SYSTEM FillerModule (* Module Filler, generated from its module specification *)
  (* Standard: 61499-2 *)
  APPLICATION Filler (* Module Filler on target pc (localhost, IO modbus; generated by modgen) *)
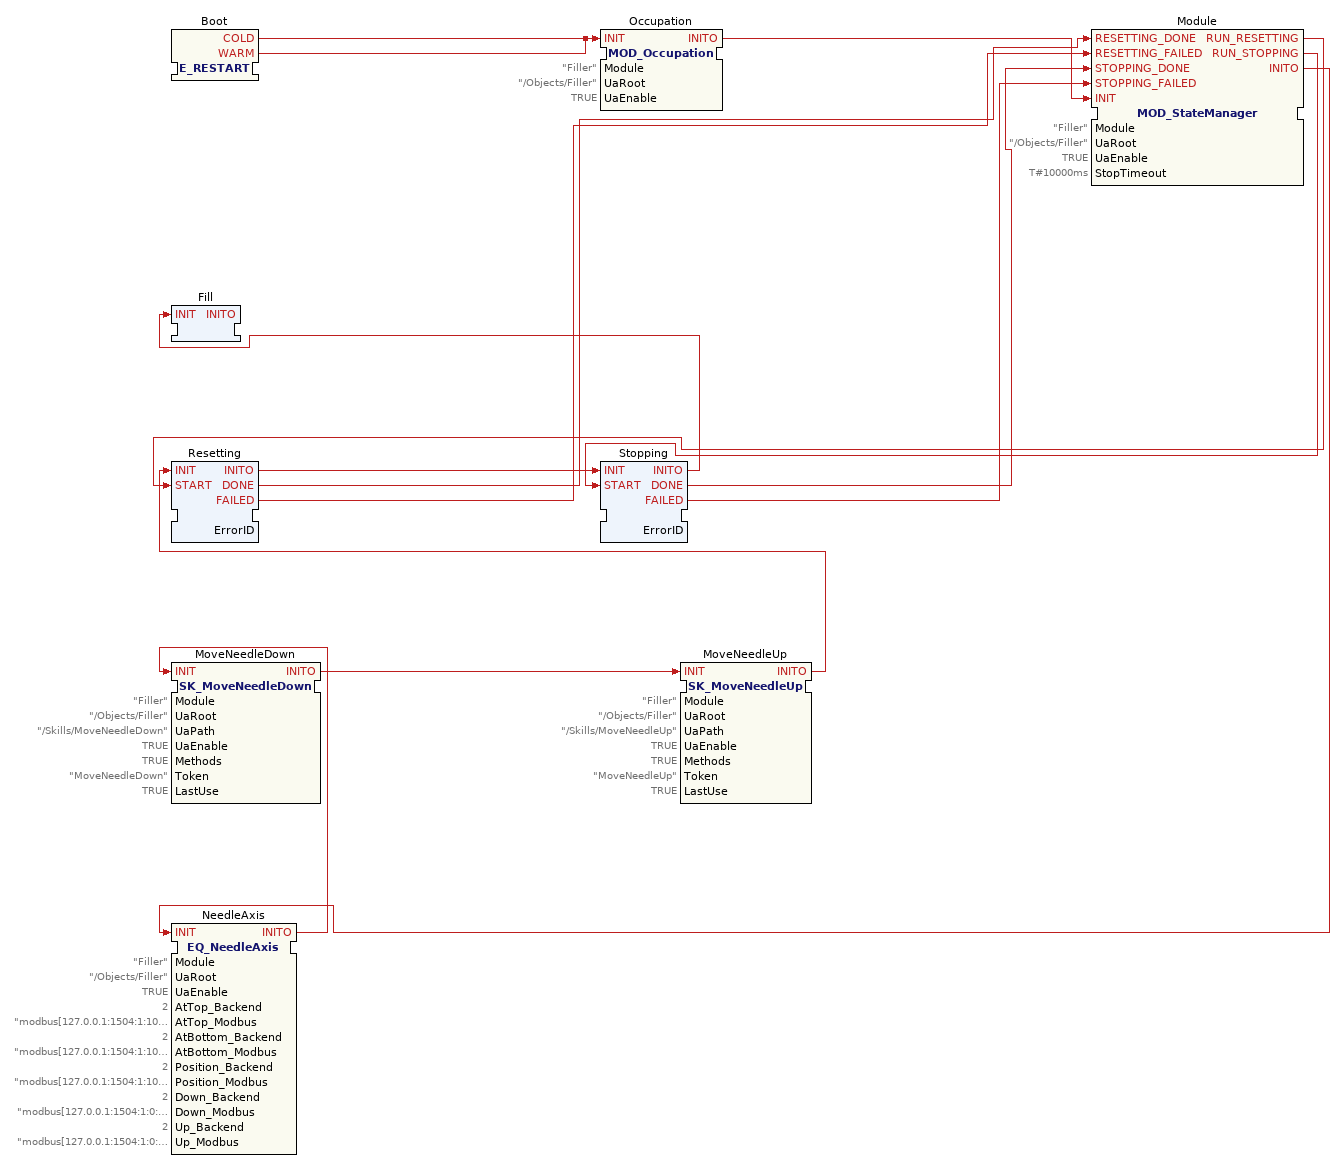
    (* Group ModuleLevel: Module level: occupation, PackML state manager, start-up and the target's IO lines *)
    (* Group ModuleLevelSkills: Module level skills: Control, Sequences (Execute, Stop) of skill primitives and Release; OPC UA /Skills/<name> *)
    (* Group Procedures: Procedures the module state manager runs while Resetting and Stopping *)
    (* Group SkillPrimitives: Skill primitives: one equipment command until a sensor or a time; OPC UA /Skills/<name> *)
    (* Group EquipmentIO: Equipment IO: the only owners of the IO points; skills send them output values over local channels *)
    FBS
      Boot : iec61499::events::E_RESTART; {SET_ATTRIBUTE(GroupName, ModuleLevel)}
      Occupation : modlib::MOD_Occupation(Module := "Filler", UaRoot := "/Objects/Filler", UaEnable := TRUE); {SET_ATTRIBUTE(GroupName, ModuleLevel)}
      Module : modlib::MOD_StateManager(Module := "Filler", UaRoot := "/Objects/Filler", UaEnable := TRUE, StopTimeout := T#10000ms); {SET_ATTRIBUTE(GroupName, ModuleLevel)}
      NeedleAxis : filler::EQ_NeedleAxis(Module := "Filler", UaRoot := "/Objects/Filler", UaEnable := TRUE, AtTop_Backend := 2, AtTop_Modbus := "modbus[127.0.0.1:1504:1:10:d0:]", AtBottom_Backend := 2, AtBottom_Modbus := "modbus[127.0.0.1:1504:1:10:d1:]", Position_Backend := 2, Position_Modbus := "modbus[127.0.0.1:1504:1:10:i1:]", Down_Backend := 2, Down_Modbus := "modbus[127.0.0.1:1504:1:0::c0]", Up_Backend := 2, Up_Modbus := "modbus[127.0.0.1:1504:1:0::c2]"); {SET_ATTRIBUTE(GroupName, EquipmentIO)}
      MoveNeedleDown : filler::SK_MoveNeedleDown(Module := "Filler", UaRoot := "/Objects/Filler", UaPath := "/Skills/MoveNeedleDown", UaEnable := TRUE, Methods := TRUE, Token := "MoveNeedleDown", LastUse := TRUE); {SET_ATTRIBUTE(GroupName, SkillPrimitives)}
      MoveNeedleUp : filler::SK_MoveNeedleUp(Module := "Filler", UaRoot := "/Objects/Filler", UaPath := "/Skills/MoveNeedleUp", UaEnable := TRUE, Methods := TRUE, Token := "MoveNeedleUp", LastUse := TRUE); {SET_ATTRIBUTE(GroupName, SkillPrimitives)}
    END_FBS
    SUBAPPLICATION Resetting (* Procedure the module runs while Resetting *)
      {SET_ATTRIBUTE(GroupName, Procedures)}
      EVENT_INPUT
        INIT : EInit;
        START;
      END_EVENT
      EVENT_OUTPUT
        INITO : EInit;
        DONE;
        FAILED;
      END_EVENT
      VAR_OUTPUT
        ErrorID : UINT;
      END_VAR
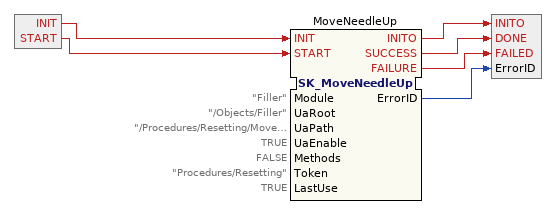
      FBS
        MoveNeedleUp : filler::SK_MoveNeedleUp(Module := "Filler", UaRoot := "/Objects/Filler", UaPath := "/Procedures/Resetting/MoveNeedleUp", UaEnable := TRUE, Methods := FALSE, Token := "Procedures/Resetting", LastUse := TRUE);
      END_FBS
      EVENT_CONNECTIONS
        INIT TO MoveNeedleUp.INIT;
        MoveNeedleUp.INITO TO INITO;
        START TO MoveNeedleUp.START;
        MoveNeedleUp.SUCCESS TO DONE;
        MoveNeedleUp.FAILURE TO FAILED;
      END_CONNECTIONS
      DATA_CONNECTIONS
        MoveNeedleUp.ErrorID TO ErrorID;
      END_CONNECTIONS
    END_SUBAPPLICATION
    SUBAPPLICATION Stopping (* Procedure the module runs while Stopping *)
      {SET_ATTRIBUTE(GroupName, Procedures)}
      EVENT_INPUT
        INIT : EInit;
        START;
      END_EVENT
      EVENT_OUTPUT
        INITO : EInit;
        DONE;
        FAILED;
      END_EVENT
      VAR_OUTPUT
        ErrorID : UINT;
      END_VAR
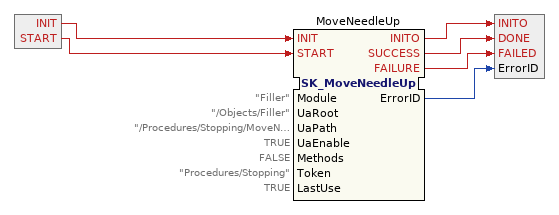
      FBS
        MoveNeedleUp : filler::SK_MoveNeedleUp(Module := "Filler", UaRoot := "/Objects/Filler", UaPath := "/Procedures/Stopping/MoveNeedleUp", UaEnable := TRUE, Methods := FALSE, Token := "Procedures/Stopping", LastUse := TRUE);
      END_FBS
      EVENT_CONNECTIONS
        INIT TO MoveNeedleUp.INIT;
        MoveNeedleUp.INITO TO INITO;
        START TO MoveNeedleUp.START;
        MoveNeedleUp.SUCCESS TO DONE;
        MoveNeedleUp.FAILURE TO FAILED;
      END_CONNECTIONS
      DATA_CONNECTIONS
        MoveNeedleUp.ErrorID TO ErrorID;
      END_CONNECTIONS
    END_SUBAPPLICATION
    SUBAPPLICATION Fill (* Module level skill Fill: Needle down to Depth and back up; a stop lifts the needle *)
      {SET_ATTRIBUTE(GroupName, ModuleLevelSkills)}
      EVENT_INPUT
        INIT : EInit;
      END_EVENT
      EVENT_OUTPUT
        INITO : EInit;
      END_EVENT
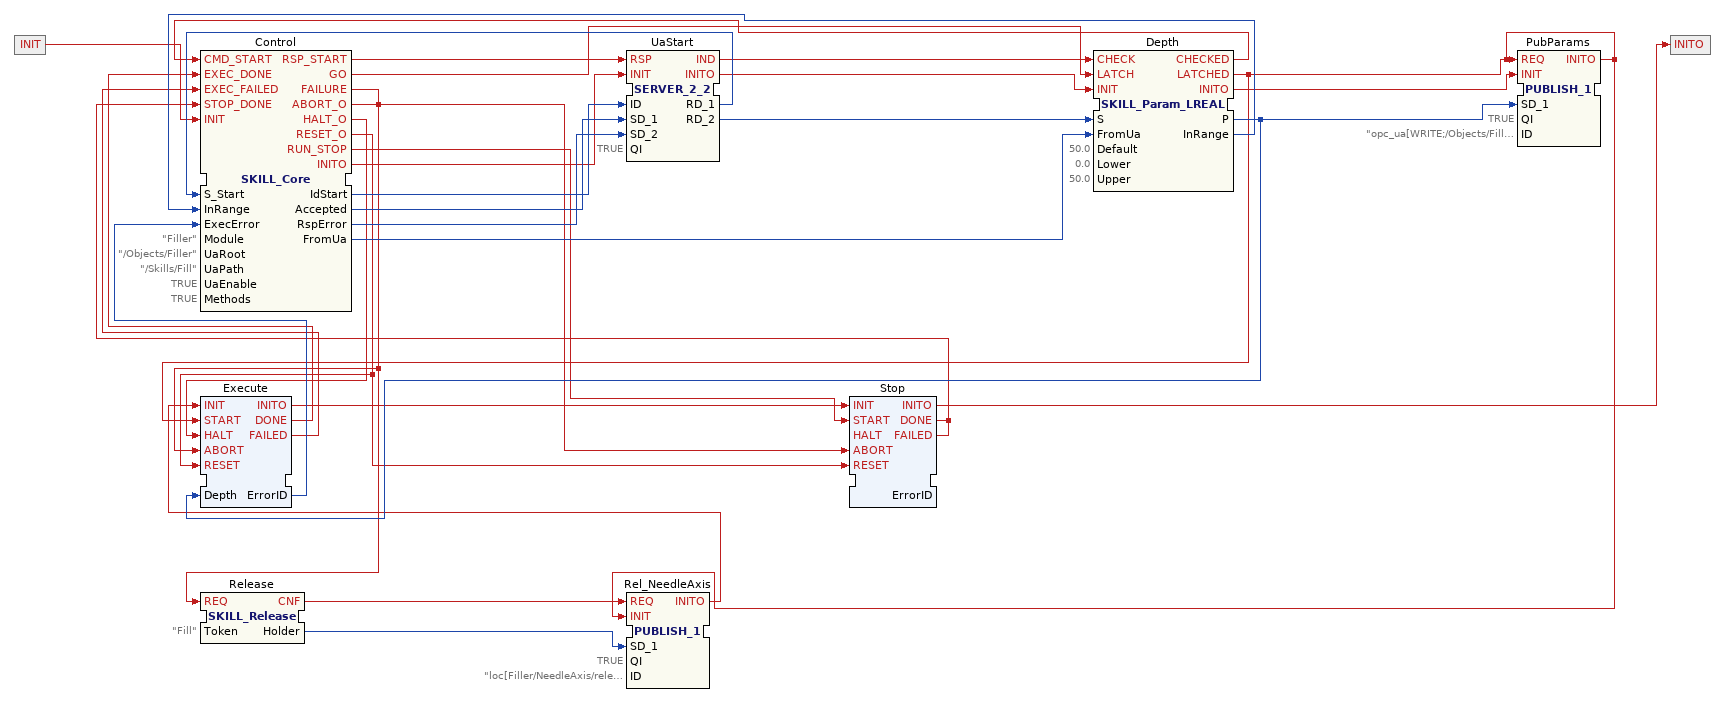
      (* Group SkillControl: State machine and OPC UA: Start(Session, parameters) with one block per parameter (range check, value for this run), Stop, Abort, Reset; State, parameters and results published *)
      (* Group Sequences: What the skill does: Execute, and Stop when it is interrupted; private skill primitives in order *)
      (* Group Releasing: After a failure or an abort: gives up the equipment the skill holds (all off, free again) *)
      FBS
        Control : modlib::SKILL_Core(Module := "Filler", UaRoot := "/Objects/Filler", UaPath := "/Skills/Fill", UaEnable := TRUE, Methods := TRUE); {SET_ATTRIBUTE(GroupName, SkillControl)}
        UaStart : iec61499::net::SERVER_2_2(QI := TRUE); {SET_ATTRIBUTE(GroupName, SkillControl)}
        Depth : modlib::SKILL_Param_LREAL(Default := 50.0, Lower := 0.0, Upper := 50.0); {SET_ATTRIBUTE(GroupName, SkillControl)}
        PubParams : iec61499::net::PUBLISH_1(QI := TRUE, ID := "opc_ua[WRITE;/Objects/Filler/Skills/Fill/Parameters/Depth]"); {SET_ATTRIBUTE(GroupName, SkillControl)}
        Release : modlib::SKILL_Release(Token := "Fill"); {SET_ATTRIBUTE(GroupName, Releasing)}
        Rel_NeedleAxis : iec61499::net::PUBLISH_1(QI := TRUE, ID := "loc[Filler/NeedleAxis/release]"); {SET_ATTRIBUTE(GroupName, Releasing)}
      END_FBS
      SUBAPPLICATION Execute (* Fill: execute sequence *)
        {SET_ATTRIBUTE(GroupName, Sequences)}
        EVENT_INPUT
          INIT : EInit;
          START;
          HALT;
          ABORT;
          RESET;
        END_EVENT
        EVENT_OUTPUT
          INITO : EInit;
          DONE;
          FAILED;
        END_EVENT
        VAR_INPUT
          Depth : LREAL;
        END_VAR
        VAR_OUTPUT
          ErrorID : UINT;
        END_VAR
        FBS
          MoveNeedleDown : filler::SK_MoveNeedleDown(Module := "Filler", UaRoot := "/Objects/Filler", UaPath := "/Skills/Fill/Execute/MoveNeedleDown", UaEnable := TRUE, Methods := FALSE, Token := "Fill", LastUse := FALSE);
          MoveNeedleUp : filler::SK_MoveNeedleUp(Module := "Filler", UaRoot := "/Objects/Filler", UaPath := "/Skills/Fill/Execute/MoveNeedleUp", UaEnable := TRUE, Methods := FALSE, Token := "Fill", LastUse := TRUE);
          Fail1 : modlib::SKILL_FailMerge;
        END_FBS
        EVENT_CONNECTIONS
          INIT TO MoveNeedleDown.INIT;
          MoveNeedleUp.INITO TO INITO;
          START TO MoveNeedleDown.START;
          MoveNeedleUp.SUCCESS TO DONE;
          MoveNeedleDown.INITO TO MoveNeedleUp.INIT;
          MoveNeedleDown.SUCCESS TO MoveNeedleUp.START;
          HALT TO MoveNeedleDown.HALT;
          HALT TO MoveNeedleUp.HALT;
          ABORT TO MoveNeedleDown.ABORT;
          ABORT TO MoveNeedleUp.ABORT;
          RESET TO MoveNeedleDown.RESET;
          RESET TO MoveNeedleUp.RESET;
          MoveNeedleDown.FAILURE TO Fail1.FAIL_A;
          MoveNeedleUp.FAILURE TO Fail1.FAIL_B;
          Fail1.FAIL TO FAILED;
        END_CONNECTIONS
        DATA_CONNECTIONS
          MoveNeedleDown.ErrorID TO Fail1.ErrA;
          MoveNeedleUp.ErrorID TO Fail1.ErrB;
          Fail1.Err TO ErrorID;
          Depth TO MoveNeedleDown.Distance;
        END_CONNECTIONS
      END_SUBAPPLICATION
      SUBAPPLICATION Stop (* Fill: stop sequence *)
        {SET_ATTRIBUTE(GroupName, Sequences)}
        EVENT_INPUT
          INIT : EInit;
          START;
          HALT;
          ABORT;
          RESET;
        END_EVENT
        EVENT_OUTPUT
          INITO : EInit;
          DONE;
          FAILED;
        END_EVENT
        VAR_OUTPUT
          ErrorID : UINT;
        END_VAR
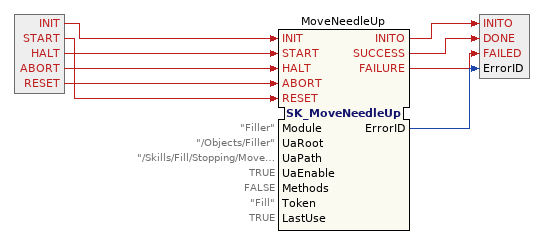
        FBS
          MoveNeedleUp : filler::SK_MoveNeedleUp(Module := "Filler", UaRoot := "/Objects/Filler", UaPath := "/Skills/Fill/Stopping/MoveNeedleUp", UaEnable := TRUE, Methods := FALSE, Token := "Fill", LastUse := TRUE);
        END_FBS
        EVENT_CONNECTIONS
          INIT TO MoveNeedleUp.INIT;
          MoveNeedleUp.INITO TO INITO;
          START TO MoveNeedleUp.START;
          MoveNeedleUp.SUCCESS TO DONE;
          HALT TO MoveNeedleUp.HALT;
          ABORT TO MoveNeedleUp.ABORT;
          RESET TO MoveNeedleUp.RESET;
          MoveNeedleUp.FAILURE TO FAILED;
        END_CONNECTIONS
        DATA_CONNECTIONS
          MoveNeedleUp.ErrorID TO ErrorID;
        END_CONNECTIONS
      END_SUBAPPLICATION
      EVENT_CONNECTIONS
        Control.RSP_START TO UaStart.RSP;
        UaStart.IND TO Depth.CHECK;
        Control.GO TO Depth.LATCH;
        Depth.CHECKED TO Control.CMD_START;
        Depth.LATCHED TO PubParams.REQ;
        PubParams.INITO TO PubParams.REQ;
        Control.FAILURE TO Release.REQ;
        Control.ABORT_O TO Release.REQ;
        Release.CNF TO Rel_NeedleAxis.REQ;
        Depth.LATCHED TO Execute.START;
        Control.HALT_O TO Execute.HALT;
        Control.ABORT_O TO Execute.ABORT;
        Control.RESET_O TO Execute.RESET;
        Execute.DONE TO Control.EXEC_DONE;
        Execute.FAILED TO Control.EXEC_FAILED;
        Control.RUN_STOP TO Stop.START;
        Control.ABORT_O TO Stop.ABORT;
        Control.RESET_O TO Stop.RESET;
        Stop.DONE TO Control.STOP_DONE;
        Stop.FAILED TO Control.STOP_DONE;
        INIT TO Control.INIT;
        Control.INITO TO UaStart.INIT;
        UaStart.INITO TO Depth.INIT;
        Depth.INITO TO PubParams.INIT;
        PubParams.INITO TO Rel_NeedleAxis.INIT;
        Rel_NeedleAxis.INITO TO Execute.INIT;
        Execute.INITO TO Stop.INIT;
        Stop.INITO TO INITO;
      END_CONNECTIONS
      DATA_CONNECTIONS
        Control.IdStart TO UaStart.ID;
        UaStart.RD_1 TO Control.S_Start;
        Control.Accepted TO UaStart.SD_1;
        Control.RspError TO UaStart.SD_2;
        UaStart.RD_2 TO Depth.S;
        Control.FromUa TO Depth.FromUa;
        Depth.P TO PubParams.SD_1;
        Depth.InRange TO Control.InRange;
        Release.Holder TO Rel_NeedleAxis.SD_1;
        Depth.P TO Execute.Depth;
        Execute.ErrorID TO Control.ExecError;
      END_CONNECTIONS
    END_SUBAPPLICATION
    EVENT_CONNECTIONS
      Boot.COLD TO Occupation.INIT;
      Boot.WARM TO Occupation.INIT;
      Module.RUN_RESETTING TO Resetting.START;
      Resetting.DONE TO Module.RESETTING_DONE;
      Resetting.FAILED TO Module.RESETTING_FAILED;
      Module.RUN_STOPPING TO Stopping.START;
      Stopping.DONE TO Module.STOPPING_DONE;
      Stopping.FAILED TO Module.STOPPING_FAILED;
      Occupation.INITO TO Module.INIT;
      Module.INITO TO NeedleAxis.INIT;
      NeedleAxis.INITO TO MoveNeedleDown.INIT;
      MoveNeedleDown.INITO TO MoveNeedleUp.INIT;
      MoveNeedleUp.INITO TO Resetting.INIT;
      Resetting.INITO TO Stopping.INIT;
      Stopping.INITO TO Fill.INIT;
    END_CONNECTIONS
  END_APPLICATION
  APPLICATION Filler_pi (* Module Filler on target pi (192.168.0.191, IO gpio; generated by modgen) *)
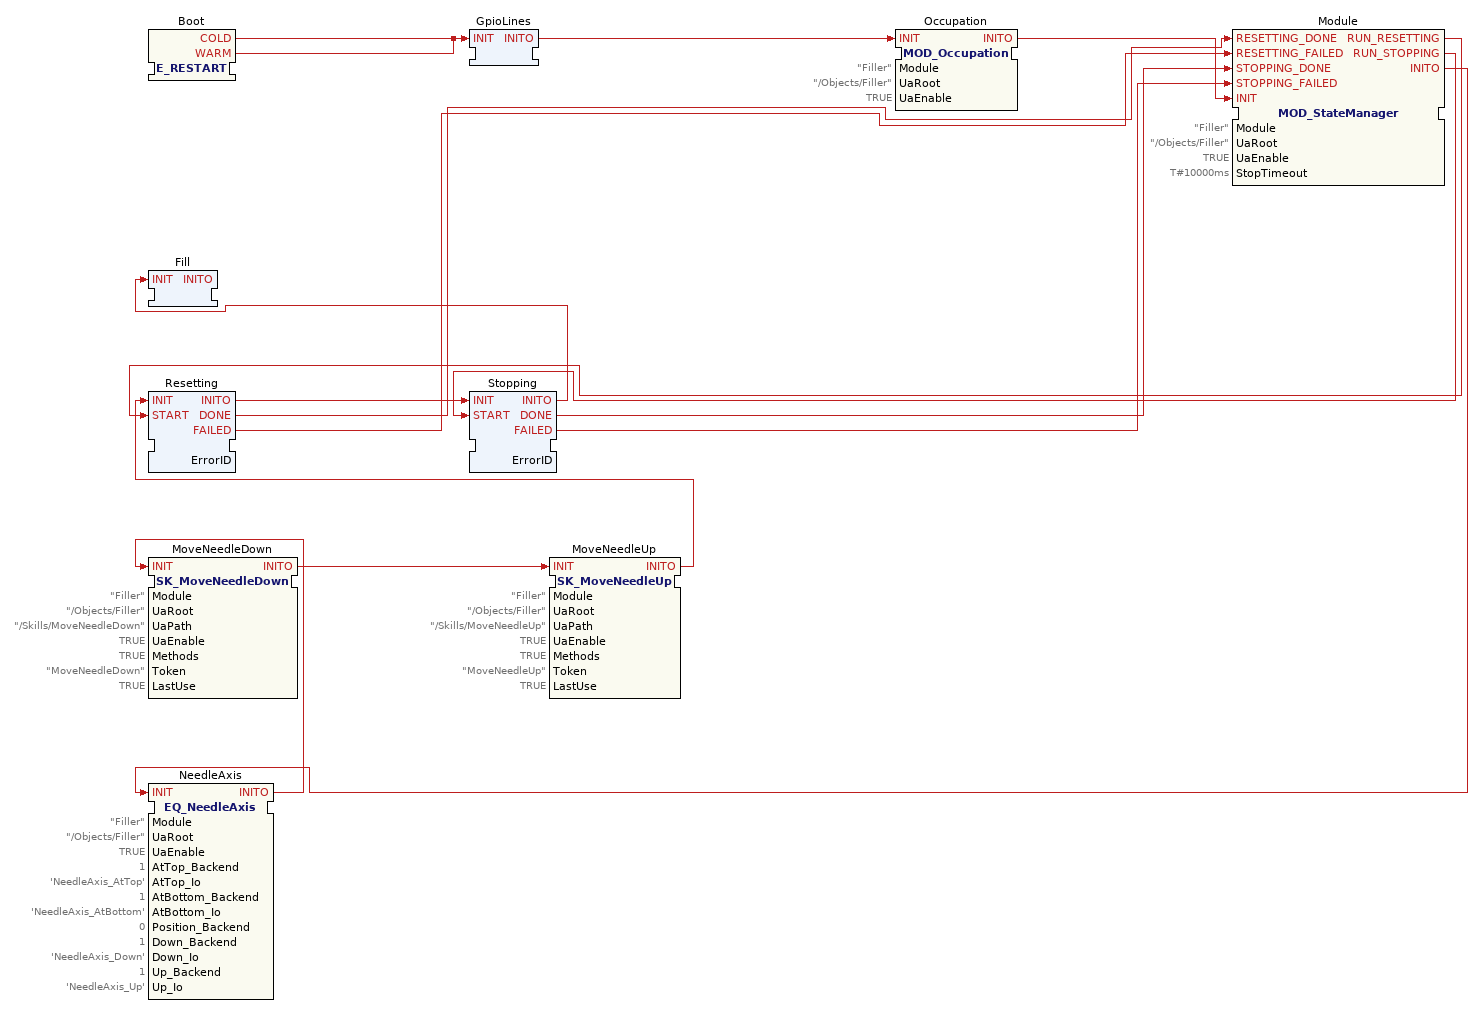
    (* Group ModuleLevel: Module level: occupation, PackML state manager, start-up and the target's IO lines *)
    (* Group ModuleLevelSkills: Module level skills: Control, Sequences (Execute, Stop) of skill primitives and Release; OPC UA /Skills/<name> *)
    (* Group Procedures: Procedures the module state manager runs while Resetting and Stopping *)
    (* Group SkillPrimitives: Skill primitives: one equipment command until a sensor or a time; OPC UA /Skills/<name> *)
    (* Group EquipmentIO: Equipment IO: the only owners of the IO points; skills send them output values over local channels *)
    FBS
      Boot : iec61499::events::E_RESTART; {SET_ATTRIBUTE(GroupName, ModuleLevel)}
      Occupation : modlib::MOD_Occupation(Module := "Filler", UaRoot := "/Objects/Filler", UaEnable := TRUE); {SET_ATTRIBUTE(GroupName, ModuleLevel)}
      Module : modlib::MOD_StateManager(Module := "Filler", UaRoot := "/Objects/Filler", UaEnable := TRUE, StopTimeout := T#10000ms); {SET_ATTRIBUTE(GroupName, ModuleLevel)}
      NeedleAxis : filler::EQ_NeedleAxis(Module := "Filler", UaRoot := "/Objects/Filler", UaEnable := TRUE, AtTop_Backend := 1, AtTop_Io := 'NeedleAxis_AtTop', AtBottom_Backend := 1, AtBottom_Io := 'NeedleAxis_AtBottom', Position_Backend := 0, Down_Backend := 1, Down_Io := 'NeedleAxis_Down', Up_Backend := 1, Up_Io := 'NeedleAxis_Up'); {SET_ATTRIBUTE(GroupName, EquipmentIO)}
      MoveNeedleDown : filler::SK_MoveNeedleDown(Module := "Filler", UaRoot := "/Objects/Filler", UaPath := "/Skills/MoveNeedleDown", UaEnable := TRUE, Methods := TRUE, Token := "MoveNeedleDown", LastUse := TRUE); {SET_ATTRIBUTE(GroupName, SkillPrimitives)}
      MoveNeedleUp : filler::SK_MoveNeedleUp(Module := "Filler", UaRoot := "/Objects/Filler", UaPath := "/Skills/MoveNeedleUp", UaEnable := TRUE, Methods := TRUE, Token := "MoveNeedleUp", LastUse := TRUE); {SET_ATTRIBUTE(GroupName, SkillPrimitives)}
    END_FBS
    SUBAPPLICATION GpioLines (* GPIO lines of the equipment's IO points (Linux /dev/gpiochip) *)
      {SET_ATTRIBUTE(GroupName, ModuleLevel)}
      EVENT_INPUT
        INIT : EInit;
      END_EVENT
      EVENT_OUTPUT
        INITO : EInit;
      END_EVENT
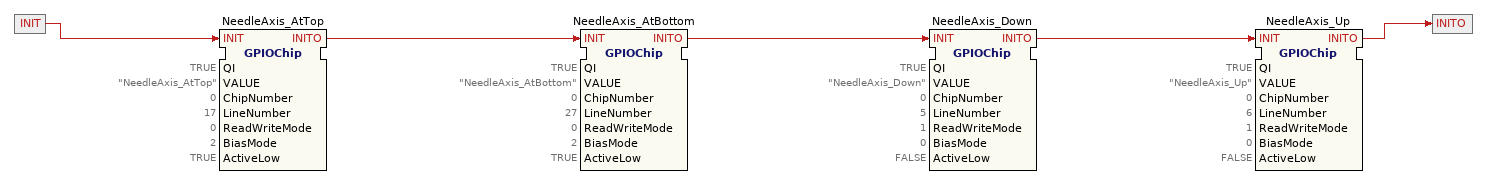
      FBS
        NeedleAxis_AtTop : eclipse4diac::io::gpiochip::GPIOChip(QI := TRUE, VALUE := "NeedleAxis_AtTop", ChipNumber := 0, LineNumber := 17, ReadWriteMode := 0, BiasMode := 2, ActiveLow := TRUE);
        NeedleAxis_AtBottom : eclipse4diac::io::gpiochip::GPIOChip(QI := TRUE, VALUE := "NeedleAxis_AtBottom", ChipNumber := 0, LineNumber := 27, ReadWriteMode := 0, BiasMode := 2, ActiveLow := TRUE);
        NeedleAxis_Down : eclipse4diac::io::gpiochip::GPIOChip(QI := TRUE, VALUE := "NeedleAxis_Down", ChipNumber := 0, LineNumber := 5, ReadWriteMode := 1, BiasMode := 0, ActiveLow := FALSE);
        NeedleAxis_Up : eclipse4diac::io::gpiochip::GPIOChip(QI := TRUE, VALUE := "NeedleAxis_Up", ChipNumber := 0, LineNumber := 6, ReadWriteMode := 1, BiasMode := 0, ActiveLow := FALSE);
      END_FBS
      EVENT_CONNECTIONS
        INIT TO NeedleAxis_AtTop.INIT;
        NeedleAxis_Up.INITO TO INITO;
        NeedleAxis_AtTop.INITO TO NeedleAxis_AtBottom.INIT;
        NeedleAxis_AtBottom.INITO TO NeedleAxis_Down.INIT;
        NeedleAxis_Down.INITO TO NeedleAxis_Up.INIT;
      END_CONNECTIONS
    END_SUBAPPLICATION
    SUBAPPLICATION Resetting (* Procedure the module runs while Resetting *)
      {SET_ATTRIBUTE(GroupName, Procedures)}
      EVENT_INPUT
        INIT : EInit;
        START;
      END_EVENT
      EVENT_OUTPUT
        INITO : EInit;
        DONE;
        FAILED;
      END_EVENT
      VAR_OUTPUT
        ErrorID : UINT;
      END_VAR
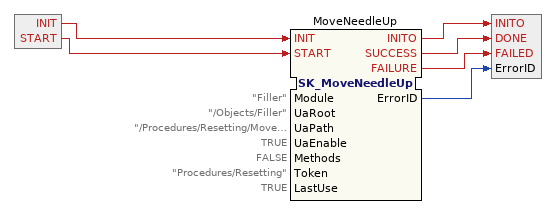
      FBS
        MoveNeedleUp : filler::SK_MoveNeedleUp(Module := "Filler", UaRoot := "/Objects/Filler", UaPath := "/Procedures/Resetting/MoveNeedleUp", UaEnable := TRUE, Methods := FALSE, Token := "Procedures/Resetting", LastUse := TRUE);
      END_FBS
      EVENT_CONNECTIONS
        INIT TO MoveNeedleUp.INIT;
        MoveNeedleUp.INITO TO INITO;
        START TO MoveNeedleUp.START;
        MoveNeedleUp.SUCCESS TO DONE;
        MoveNeedleUp.FAILURE TO FAILED;
      END_CONNECTIONS
      DATA_CONNECTIONS
        MoveNeedleUp.ErrorID TO ErrorID;
      END_CONNECTIONS
    END_SUBAPPLICATION
    SUBAPPLICATION Stopping (* Procedure the module runs while Stopping *)
      {SET_ATTRIBUTE(GroupName, Procedures)}
      EVENT_INPUT
        INIT : EInit;
        START;
      END_EVENT
      EVENT_OUTPUT
        INITO : EInit;
        DONE;
        FAILED;
      END_EVENT
      VAR_OUTPUT
        ErrorID : UINT;
      END_VAR
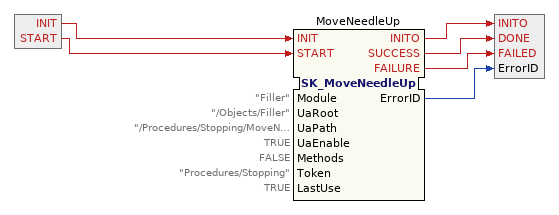
      FBS
        MoveNeedleUp : filler::SK_MoveNeedleUp(Module := "Filler", UaRoot := "/Objects/Filler", UaPath := "/Procedures/Stopping/MoveNeedleUp", UaEnable := TRUE, Methods := FALSE, Token := "Procedures/Stopping", LastUse := TRUE);
      END_FBS
      EVENT_CONNECTIONS
        INIT TO MoveNeedleUp.INIT;
        MoveNeedleUp.INITO TO INITO;
        START TO MoveNeedleUp.START;
        MoveNeedleUp.SUCCESS TO DONE;
        MoveNeedleUp.FAILURE TO FAILED;
      END_CONNECTIONS
      DATA_CONNECTIONS
        MoveNeedleUp.ErrorID TO ErrorID;
      END_CONNECTIONS
    END_SUBAPPLICATION
    SUBAPPLICATION Fill (* Module level skill Fill: Needle down to Depth and back up; a stop lifts the needle *)
      {SET_ATTRIBUTE(GroupName, ModuleLevelSkills)}
      EVENT_INPUT
        INIT : EInit;
      END_EVENT
      EVENT_OUTPUT
        INITO : EInit;
      END_EVENT
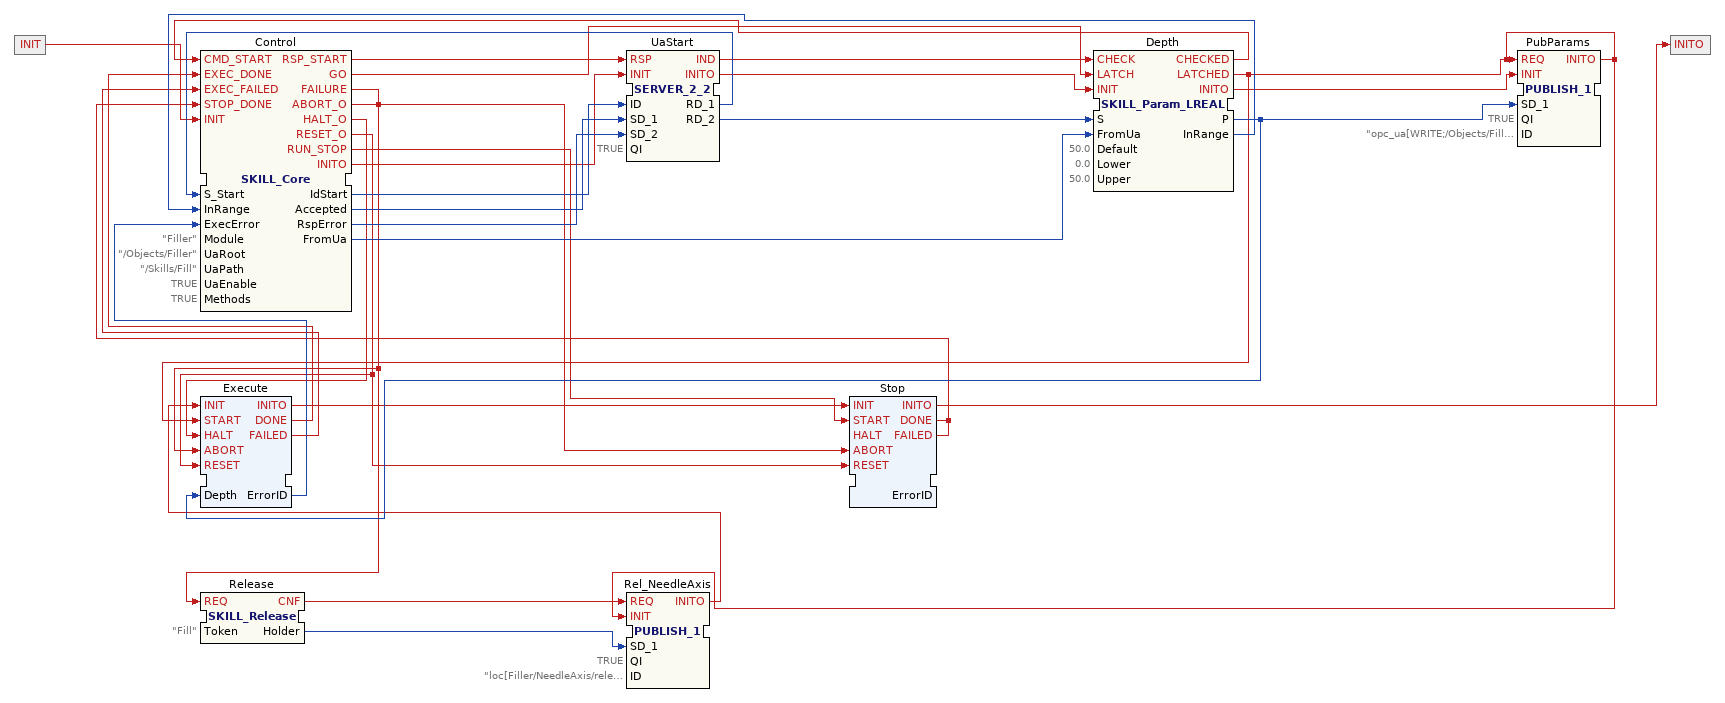
      (* Group SkillControl: State machine and OPC UA: Start(Session, parameters) with one block per parameter (range check, value for this run), Stop, Abort, Reset; State, parameters and results published *)
      (* Group Sequences: What the skill does: Execute, and Stop when it is interrupted; private skill primitives in order *)
      (* Group Releasing: After a failure or an abort: gives up the equipment the skill holds (all off, free again) *)
      FBS
        Control : modlib::SKILL_Core(Module := "Filler", UaRoot := "/Objects/Filler", UaPath := "/Skills/Fill", UaEnable := TRUE, Methods := TRUE); {SET_ATTRIBUTE(GroupName, SkillControl)}
        UaStart : iec61499::net::SERVER_2_2(QI := TRUE); {SET_ATTRIBUTE(GroupName, SkillControl)}
        Depth : modlib::SKILL_Param_LREAL(Default := 50.0, Lower := 0.0, Upper := 50.0); {SET_ATTRIBUTE(GroupName, SkillControl)}
        PubParams : iec61499::net::PUBLISH_1(QI := TRUE, ID := "opc_ua[WRITE;/Objects/Filler/Skills/Fill/Parameters/Depth]"); {SET_ATTRIBUTE(GroupName, SkillControl)}
        Release : modlib::SKILL_Release(Token := "Fill"); {SET_ATTRIBUTE(GroupName, Releasing)}
        Rel_NeedleAxis : iec61499::net::PUBLISH_1(QI := TRUE, ID := "loc[Filler/NeedleAxis/release]"); {SET_ATTRIBUTE(GroupName, Releasing)}
      END_FBS
      SUBAPPLICATION Execute (* Fill: execute sequence *)
        {SET_ATTRIBUTE(GroupName, Sequences)}
        EVENT_INPUT
          INIT : EInit;
          START;
          HALT;
          ABORT;
          RESET;
        END_EVENT
        EVENT_OUTPUT
          INITO : EInit;
          DONE;
          FAILED;
        END_EVENT
        VAR_INPUT
          Depth : LREAL;
        END_VAR
        VAR_OUTPUT
          ErrorID : UINT;
        END_VAR
        FBS
          MoveNeedleDown : filler::SK_MoveNeedleDown(Module := "Filler", UaRoot := "/Objects/Filler", UaPath := "/Skills/Fill/Execute/MoveNeedleDown", UaEnable := TRUE, Methods := FALSE, Token := "Fill", LastUse := FALSE);
          MoveNeedleUp : filler::SK_MoveNeedleUp(Module := "Filler", UaRoot := "/Objects/Filler", UaPath := "/Skills/Fill/Execute/MoveNeedleUp", UaEnable := TRUE, Methods := FALSE, Token := "Fill", LastUse := TRUE);
          Fail1 : modlib::SKILL_FailMerge;
        END_FBS
        EVENT_CONNECTIONS
          INIT TO MoveNeedleDown.INIT;
          MoveNeedleUp.INITO TO INITO;
          START TO MoveNeedleDown.START;
          MoveNeedleUp.SUCCESS TO DONE;
          MoveNeedleDown.INITO TO MoveNeedleUp.INIT;
          MoveNeedleDown.SUCCESS TO MoveNeedleUp.START;
          HALT TO MoveNeedleDown.HALT;
          HALT TO MoveNeedleUp.HALT;
          ABORT TO MoveNeedleDown.ABORT;
          ABORT TO MoveNeedleUp.ABORT;
          RESET TO MoveNeedleDown.RESET;
          RESET TO MoveNeedleUp.RESET;
          MoveNeedleDown.FAILURE TO Fail1.FAIL_A;
          MoveNeedleUp.FAILURE TO Fail1.FAIL_B;
          Fail1.FAIL TO FAILED;
        END_CONNECTIONS
        DATA_CONNECTIONS
          MoveNeedleDown.ErrorID TO Fail1.ErrA;
          MoveNeedleUp.ErrorID TO Fail1.ErrB;
          Fail1.Err TO ErrorID;
          Depth TO MoveNeedleDown.Distance;
        END_CONNECTIONS
      END_SUBAPPLICATION
      SUBAPPLICATION Stop (* Fill: stop sequence *)
        {SET_ATTRIBUTE(GroupName, Sequences)}
        EVENT_INPUT
          INIT : EInit;
          START;
          HALT;
          ABORT;
          RESET;
        END_EVENT
        EVENT_OUTPUT
          INITO : EInit;
          DONE;
          FAILED;
        END_EVENT
        VAR_OUTPUT
          ErrorID : UINT;
        END_VAR
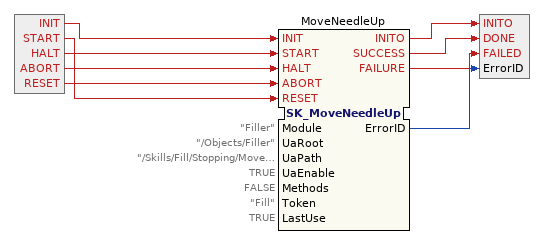
        FBS
          MoveNeedleUp : filler::SK_MoveNeedleUp(Module := "Filler", UaRoot := "/Objects/Filler", UaPath := "/Skills/Fill/Stopping/MoveNeedleUp", UaEnable := TRUE, Methods := FALSE, Token := "Fill", LastUse := TRUE);
        END_FBS
        EVENT_CONNECTIONS
          INIT TO MoveNeedleUp.INIT;
          MoveNeedleUp.INITO TO INITO;
          START TO MoveNeedleUp.START;
          MoveNeedleUp.SUCCESS TO DONE;
          HALT TO MoveNeedleUp.HALT;
          ABORT TO MoveNeedleUp.ABORT;
          RESET TO MoveNeedleUp.RESET;
          MoveNeedleUp.FAILURE TO FAILED;
        END_CONNECTIONS
        DATA_CONNECTIONS
          MoveNeedleUp.ErrorID TO ErrorID;
        END_CONNECTIONS
      END_SUBAPPLICATION
      EVENT_CONNECTIONS
        Control.RSP_START TO UaStart.RSP;
        UaStart.IND TO Depth.CHECK;
        Control.GO TO Depth.LATCH;
        Depth.CHECKED TO Control.CMD_START;
        Depth.LATCHED TO PubParams.REQ;
        PubParams.INITO TO PubParams.REQ;
        Control.FAILURE TO Release.REQ;
        Control.ABORT_O TO Release.REQ;
        Release.CNF TO Rel_NeedleAxis.REQ;
        Depth.LATCHED TO Execute.START;
        Control.HALT_O TO Execute.HALT;
        Control.ABORT_O TO Execute.ABORT;
        Control.RESET_O TO Execute.RESET;
        Execute.DONE TO Control.EXEC_DONE;
        Execute.FAILED TO Control.EXEC_FAILED;
        Control.RUN_STOP TO Stop.START;
        Control.ABORT_O TO Stop.ABORT;
        Control.RESET_O TO Stop.RESET;
        Stop.DONE TO Control.STOP_DONE;
        Stop.FAILED TO Control.STOP_DONE;
        INIT TO Control.INIT;
        Control.INITO TO UaStart.INIT;
        UaStart.INITO TO Depth.INIT;
        Depth.INITO TO PubParams.INIT;
        PubParams.INITO TO Rel_NeedleAxis.INIT;
        Rel_NeedleAxis.INITO TO Execute.INIT;
        Execute.INITO TO Stop.INIT;
        Stop.INITO TO INITO;
      END_CONNECTIONS
      DATA_CONNECTIONS
        Control.IdStart TO UaStart.ID;
        UaStart.RD_1 TO Control.S_Start;
        Control.Accepted TO UaStart.SD_1;
        Control.RspError TO UaStart.SD_2;
        UaStart.RD_2 TO Depth.S;
        Control.FromUa TO Depth.FromUa;
        Depth.P TO PubParams.SD_1;
        Depth.InRange TO Control.InRange;
        Release.Holder TO Rel_NeedleAxis.SD_1;
        Depth.P TO Execute.Depth;
        Execute.ErrorID TO Control.ExecError;
      END_CONNECTIONS
    END_SUBAPPLICATION
    EVENT_CONNECTIONS
      Boot.COLD TO GpioLines.INIT;
      Boot.WARM TO GpioLines.INIT;
      Module.RUN_RESETTING TO Resetting.START;
      Resetting.DONE TO Module.RESETTING_DONE;
      Resetting.FAILED TO Module.RESETTING_FAILED;
      Module.RUN_STOPPING TO Stopping.START;
      Stopping.DONE TO Module.STOPPING_DONE;
      Stopping.FAILED TO Module.STOPPING_FAILED;
      GpioLines.INITO TO Occupation.INIT;
      Occupation.INITO TO Module.INIT;
      Module.INITO TO NeedleAxis.INIT;
      NeedleAxis.INITO TO MoveNeedleDown.INIT;
      MoveNeedleDown.INITO TO MoveNeedleUp.INIT;
      MoveNeedleUp.INITO TO Resetting.INIT;
      Resetting.INITO TO Stopping.INIT;
      Stopping.INITO TO Fill.INIT;
    END_CONNECTIONS
  END_APPLICATION
  DEVICE FORTE_PC : iec61499::system::FORTE_PC(MGR_ID := "localhost:61499" (* Device manager socket ID *))
    {SET_ATTRIBUTE(Profile, HOLOBLOC)}
    RESOURCE RES : iec61499::system::EMB_RES
    END_RESOURCE
  END_DEVICE
  DEVICE FORTE_PI : iec61499::system::FORTE_PC(MGR_ID := "192.168.0.191:61499" (* Device manager socket ID *))
    {SET_ATTRIBUTE(Profile, HOLOBLOC)}
    RESOURCE RES : iec61499::system::EMB_RES
    END_RESOURCE
  END_DEVICE
  MAPPINGS
    Filler.Boot ON FORTE_PC.RES;
    Filler.Occupation ON FORTE_PC.RES;
    Filler.Module ON FORTE_PC.RES;
    Filler.NeedleAxis ON FORTE_PC.RES;
    Filler.MoveNeedleDown ON FORTE_PC.RES;
    Filler.MoveNeedleUp ON FORTE_PC.RES;
    Filler.Resetting ON FORTE_PC.RES;
    Filler.Stopping ON FORTE_PC.RES;
    Filler.Fill ON FORTE_PC.RES;
    Filler_pi.Boot ON FORTE_PI.RES;
    Filler_pi.Occupation ON FORTE_PI.RES;
    Filler_pi.Module ON FORTE_PI.RES;
    Filler_pi.GpioLines ON FORTE_PI.RES;
    Filler_pi.NeedleAxis ON FORTE_PI.RES;
    Filler_pi.MoveNeedleDown ON FORTE_PI.RES;
    Filler_pi.MoveNeedleUp ON FORTE_PI.RES;
    Filler_pi.Resetting ON FORTE_PI.RES;
    Filler_pi.Stopping ON FORTE_PI.RES;
    Filler_pi.Fill ON FORTE_PI.RES;
  END_MAPPINGS
END_SYSTEM
